// Mitsubishi GX Works2 project: 20240115_AI机程序   PLC: FX3S

PROGRAM MAIN
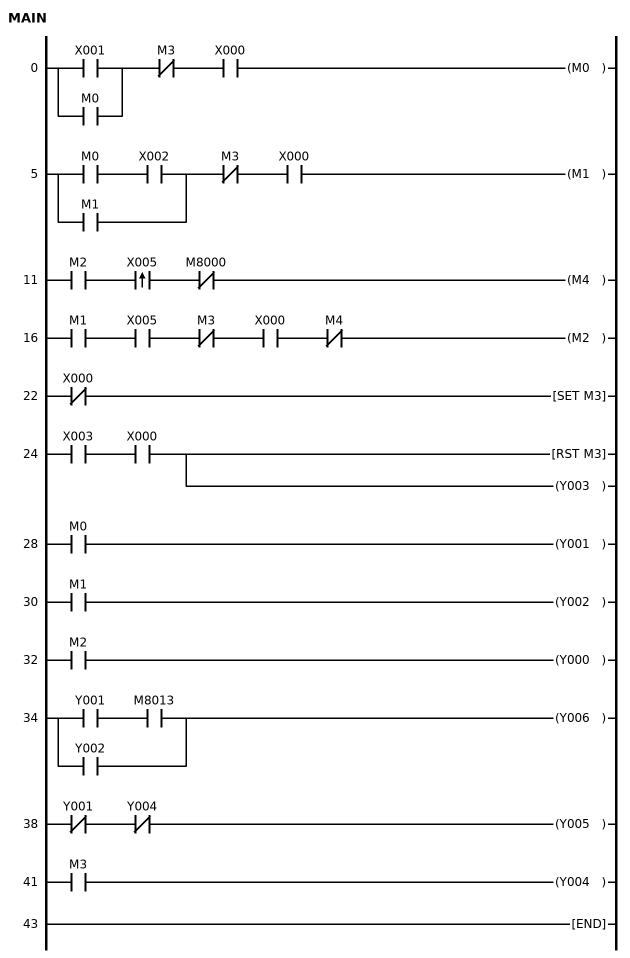
0     LD      X001
      OR      M0
      ANI     M3
      AND     X000
      OUT     M0
5     LD      M0
      AND     X002
      OR      M1
      ANI     M3
      AND     X000
      OUT     M1
11    LD      M2
      ANDP    X005
      ANI     M8000
      OUT     M4
16    LD      M1
      AND     X005
      ANI     M3
      AND     X000
      ANI     M4
      OUT     M2
22    LDI     X000
      SET     M3
24    LD      X003
      AND     X000
      RST     M3
      OUT     Y003
28    LD      M0
      OUT     Y001
30    LD      M1
      OUT     Y002
32    LD      M2
      OUT     Y000
34    LD      Y001
      AND     M8013
      OR      Y002
      OUT     Y006
38    LDI     Y001
      ANI     Y004
      OUT     Y005
41    LD      M3
      OUT     Y004
43    END
END_PROGRAM
